(* Logix 5000 project; controller ICA19 vendor 1 type 14 code 150 rev 37.11; software revision 37.00 *)

TASK MainTask (continuous, watchdog 500 ms) : MainProgram

MODULES
   Local : vendor 1 type 14 code 150 (Compact 0, rev 37.11)
      Discrete_IO : Embedded (Compact 1, rev 3.1, Output RPI 20 ms)
      Analog_IO : Embedded (Compact 2, rev 1.1, Output RPI 80 ms)
      Counters : Embedded (Compact 3, rev 1.1, Output RPI 20 ms)
END_MODULES

VAR_GLOBAL   (* controller tags *)
   DoorClosed : STRING;
   DoorOpening : STRING;
   MotorDOWN : BOOL;
   MotorUP : BOOL;
   SEQ : DINT;
   TopBottom : BOOL;
   TopLimit : BOOL;
END_VAR

PROGRAM MainProgram   (* main routine MainRoutine *)

ROUTINE Main_Status   (* ladder *)
   0: ;
END_ROUTINE

ROUTINE MainRoutine   (* ladder *)
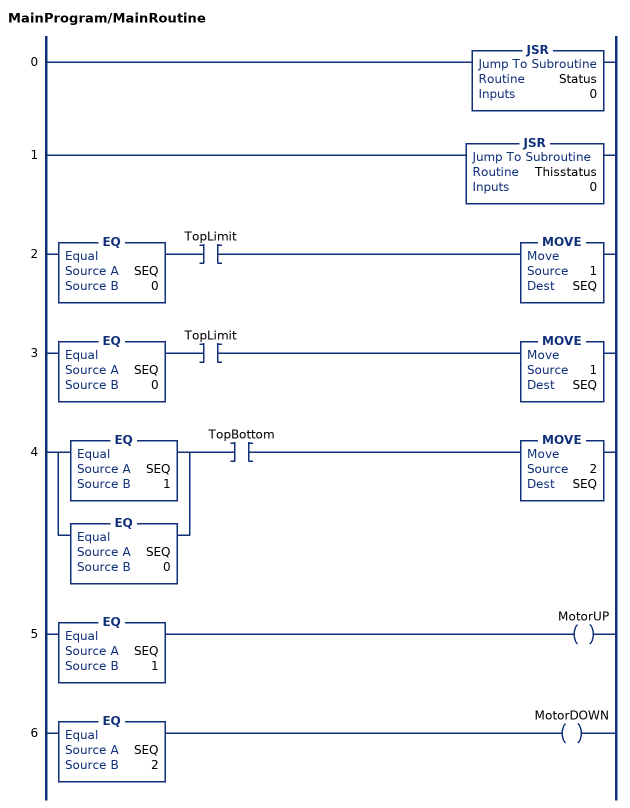
   0: JSR(Status,0);
   1: JSR(Thisstatus,0);
   2: EQ(SEQ,0)XIC(TopLimit)MOVE(1,SEQ);
   3: EQ(SEQ,0)XIC(TopLimit)MOVE(1,SEQ);
   4: [EQ(SEQ,1) ,EQ(SEQ,0) ]XIC(TopBottom)MOVE(2,SEQ);
   5: EQ(SEQ,1)OTE(MotorUP);
   6: EQ(SEQ,2)OTE(MotorDOWN);
END_ROUTINE

ROUTINE Status   (* structured text *)
   if SEQ=0 then
   	concat(
END_ROUTINE

ROUTINE Thisstatus   (* structured text *)
   if SEQ = 0 then
   
END_ROUTINE
END_PROGRAM
